// TIA Portal V20 export
TYPE "LBP_typeMcp483StandardOutput"
TITLE = MCP 483 image / Image du MCP 483
// Output image of MCP 483 / Image de sortie du MCP 483
   STRUCT
      LEDauto : Bool;
      LEDmda : Bool;
      LEDteachIn : Bool;
      LEDjog : Bool;
      LEDinc1 : Bool;
      LEDinc10 : Bool;
      LEDinc100 : Bool;
      LEDinc1000 : Bool;
      LEDinc10000 : Bool;
      LEDincVar : Bool;
      LEDrefPoint : Bool;
      LEDrepos : Bool;
      LEDcycleStop : Bool;
      LEDcycleStart : Bool;
      LEDfeedrateStop : Bool;
      LEDfeedrateStart : Bool;
      LEDspindleStop : Bool;
      LEDspindleStart : Bool;
      LEDsingleBlock : Bool;
      LEDaxis10 : Bool;   // R10
      LEDaxis7 : Bool;   // R7
      LEDaxis4 : Bool;   // R4
      LEDaxisX : Bool;   // R1
      LEDminus : Bool;   // R13
      LEDplus : Bool;   // R15
      LEDaxis6 : Bool;   // R6
      LEDaxis8 : Bool;   // R8
      LEDaxis9 : Bool;   // R9
      LEDaxis11 : Bool;   // R11
      LEDmcsWcs : Bool;   // R12
      LEDaxis5 : Bool;   // R5
      LEDaxisZ : Bool;   // R3
      LEDaxisY : Bool;   // R2
      LEDcustomerKey15 : Bool;   // T15
      LEDcustomerKey14 : Bool;   // T14
      LEDcustomerKey13 : Bool;   // T13
      LEDcustomerKey12 : Bool;   // T12
      LEDcustomerKey11 : Bool;   // T11
      LEDcustomerKey10 : Bool;   // T10
      LEDcustomerKey9 : Bool;   // T9
      LEDcustomerKey8 : Bool;   // T8
      LEDcustomerKey7 : Bool;   // T7
      LEDcustomerKey6 : Bool;   // T6
      LEDcustomerKey5 : Bool;   // T5
      LEDcustomerKey4 : Bool;   // T4
      LEDcustomerKey3 : Bool;   // T3
      LEDcustomerKey2 : Bool;   // T2
      LEDcustomerKey1 : Bool;   // T1
      LEDrapidTraverse : Bool;   // R14
      LEDreset : Bool;
      reserved62 : Bool;
      reserved63 : Bool;
      reserved64 : Bool;
      reserved65 : Bool;
      reserved66 : Bool;
      reserved67 : Bool;
      LEDoptionalKey1 : Bool;   // KT-OUT1, reserved / KT-OUT1, réservé
      LEDoptionalKey2 : Bool;   // KT-OUT2, reserved / KT-OUT2, réservé
      LEDoptionalKey3 : Bool;   // KT-OUT3, reserved / KT-OUT3, réservé
      LEDoptionalKey4 : Bool;   // KT-OUT4, reserved / KT-OUT4, réservé
      LEDoptionalKey5 : Bool;   // KT-OUT5, reserved / KT-OUT5, réservé
      LEDoptionalKey6 : Bool;   // KT-OUT6, reserved / KT-OUT6, réservé
      reserved76 : Bool;
      reserved77 : Bool;
   END_STRUCT;
END_TYPE
